// TIA Portal V17 export
// export: Created 2022-04-06T07:28:39.6757518Z, ExportSetting WithDefaults, DisplayName Totally Integrated Automation Portal, DisplayVersion V17, DisplayName TIA Portal Openness, DisplayVersion V17, DisplayName TIA Portal Version Control Interface, DisplayVersion V17, DisplayName TIA Portal Test Suite Advanced, DisplayVersion V17, DisplayName SINAMICS Startdrive Advanced, DisplayVersion V17, DisplayName SINAMICS Startdrive G130, G150, S120, S150, SINAMICS MV, S210, DisplayVersion V17, DisplayName SINAMICS Startdrive G110M, G120, G120C, G120D, G120P, G115D, DisplayVersion V17, DisplayName STEP 7 Professional, DisplayVersion V17, DisplayName STEP 7 Safety, DisplayVersion V17, DisplayName WinCC Advanced / Unified PC, DisplayVersion V17
DATA_BLOCK "Test"   // DB4
{ S7_Optimized_Access := 'TRUE' }
VERSION : 0.1
// stored: AutoNumber true, DBAccessibleFromOPCUA true, DBAccessibleFromWebserver true, IsOnlyStoredInLoadMemory false, IsRetainMemResEnabled false, IsWriteProtectedInAS false, MemoryReserve 100
   VAR
      stoAxis1 : Bool := 1;
      stoAxis2 : Bool := 1;
      ss1Axis1 : Bool := 1;
      reset : Bool;
      reintegration : Bool;
      ss1Axis2 : Bool := 1;
      enableAxis1 : Bool;
      enableAxis2 : Bool;
      moveVelocityAxis1 : Bool;
      moveVelocityAxis2 : Bool;
      homeAxis1 : Bool;
      configAxis1 : "LAxisCtrl_typeAxisConfig";
      configAxis2 { S7_SetPoint := 'True'} : "LAxisCtrl_typeAxisConfig";
      "jog+" { S7_SetPoint := 'True'} : Bool;
      "jog-" : Bool;
      stop : Bool;
      sto1 : Bool := 1;
      sto2 : Bool := 1;
      ss2Axis1 : Bool := 1;
      ss2Axis2 : Bool := 1;
      test : Bool := 0;
      fifo : "typeFifo";
      "name" { S7_SetPoint := 'True'} : Array[0..50] of String;
      name1 : String;
      "real" : Real;
      releaseEstop : Bool := true;
      releaseGate : Bool := true;
      enableMode : Bool := 0;
      stoActiveAxis1 : Bool;
      stoActiveAxis2 : Bool;
      ss1ActiveAxis1 : Bool;
      ss1ActiveAxis2 : Bool;
      ss2ActiveAxis1 : Bool;
      ss2ActiveAxis2 : Bool;
      slsActiveAxis1 : Bool;
      slsActiveAxis2 : Bool;
   END_VAR
BEGIN
   configAxis1.moveVelocity.velocity := 40.0;
   configAxis2.moveVelocity.velocity := 40.0;
END_DATA_BLOCK
